FUNCTION_BLOCK PUBLIC FB_Matrix4x4 EXTENDS ExternalStaticMatrix
VAR_INPUT
END_VAR
VAR_OUTPUT
END_VAR
VAR
	data_array : ARRAY [0..15] OF LREAL;
END_VAR

METHOD FB_init : BOOL
VAR_INPUT
	bInitRetains : BOOL; // if TRUE, the retain variables are initialized (warm start / cold start)
	bInCopyCode : BOOL;  // if TRUE, the instance afterwards gets moved into the copy code (online change)
END_VAR
VAR
END_VAR
Init(ADR(data_array), 4, 4);
Clear();
END_METHOD

END_FUNCTION_BLOCK

(* stored: Version 1.1.0.1, ProductVersion 3.1.4024.9
   POU FB_Matrix4x4: Id {f4a9e808-a4c0-4a90-8187-6ad211a90c89}, SpecialFunc None
   Method FB_init: Id {f12619f9-cf19-4eaa-9b1a-bbbfc7ecfb01} *)
